// TIA Portal project "ATS Motor Start" (V17)

(* hardware
DEVICE "S7-1200 station_1"  S7-1200 Station
   slot 0: "Rack_0"  S7-1200 Rack  Rack  V1.0
   slot 1: "PLC_2"  CPU 1215C DC/DC/Rly  6ES7 215-1HG40-0XB0  V4.5
*)

// ===== PLC "PLC_2"  CPU 1215C DC/DC/Rly =====

VAR_GLOBAL   // PLC tag table "Default tag table"
   "Clock_Byte" AT %MB0 : Byte;
   "Clock_10Hz" AT %M0.0 : Bool;
   "Clock_5Hz" AT %M0.1 : Bool;
   "Clock_2.5Hz" AT %M0.2 : Bool;
   "Clock_2Hz" AT %M0.3 : Bool;
   "Clock_1.25Hz" AT %M0.4 : Bool;
   "Clock_1Hz" AT %M0.5 : Bool;
   "Clock_0.625Hz" AT %M0.6 : Bool;
   "Clock_0.5Hz" AT %M0.7 : Bool;
   "Tag_1" AT %M2.6 : Bool;
END_VAR

VAR_GLOBAL   // PLC tag table "Tag table_1"
   "emergency_Stop" AT %I0.0 : Bool;
   "Stop" AT %I0.1 : Bool;
   "Start" AT %I0.2 : Bool;
   "PID_Contact" AT %I0.3 : Bool;
   "R1" AT %I0.4 : Bool;
   "R2" AT %I0.5 : Bool;
   "R3" AT %I0.6 : Bool;
   "R4" AT %I0.7 : Bool;
   "R5" AT %I1.0 : Bool;
   "R6" AT %I1.1 : Bool;
   "Thermal_overload" AT %I1.2 : Bool;
   "System_ON" AT %M2.0 : Bool;
   "Backup_supply" AT %Q0.5 : Bool;
   "Main_supply" AT %Q0.6 : Bool;
   "main_k1" AT %Q0.7 : Bool;
   "Star" AT %Q1.0 : Bool;
   "Delta" AT %Q1.1 : Bool;
   "Ats_on" AT %M2.2 : Bool;
   "blue_lamp" AT %Q0.0 : Bool;
   "Green_lamp" AT %Q0.1 : Bool;
   "Red_lamp" AT %Q0.2 : Bool;
   "Yellow_lamp" AT %Q0.3 : Bool;
   "Yellow_lamp_2" AT %Q0.4 : Bool;
   "main_supply_ok" AT %M2.3 : Bool;
   "back_up_ok" AT %M2.4 : Bool;
END_VAR

// folder: System blocks/Program resources

DATA_BLOCK "IEC_Timer_0_DB"   // DB1
{ S7_Optimized_Access := 'TRUE' }
AUTHOR : Simatic
FAMILY : IEC
NAME : IEC_TMR
VERSION : 1.0
// stored: InstanceOfName IEC_TIMER
"IEC_TIMER"
BEGIN
END_DATA_BLOCK

DATA_BLOCK "IEC_Timer_0_DB_2"   // DB3
{ S7_Optimized_Access := 'TRUE' }
AUTHOR : Simatic
FAMILY : IEC
NAME : IEC_TMR
VERSION : 1.0
// stored: InstanceOfName IEC_TIMER
"IEC_TIMER"
BEGIN
END_DATA_BLOCK

DATA_BLOCK "IEC_Timer_0_DB_3"   // DB4
{ S7_Optimized_Access := 'TRUE' }
AUTHOR : Simatic
FAMILY : IEC
NAME : IEC_TMR
VERSION : 1.0
// stored: InstanceOfName IEC_TIMER
"IEC_TIMER"
BEGIN
END_DATA_BLOCK

// folder: (top level)

FUNCTION "Change_over" : Void   // FC1, LAD
{ S7_Optimized_Access := 'TRUE' }
VERSION : 0.1
BEGIN

REGION Network 1: Start system
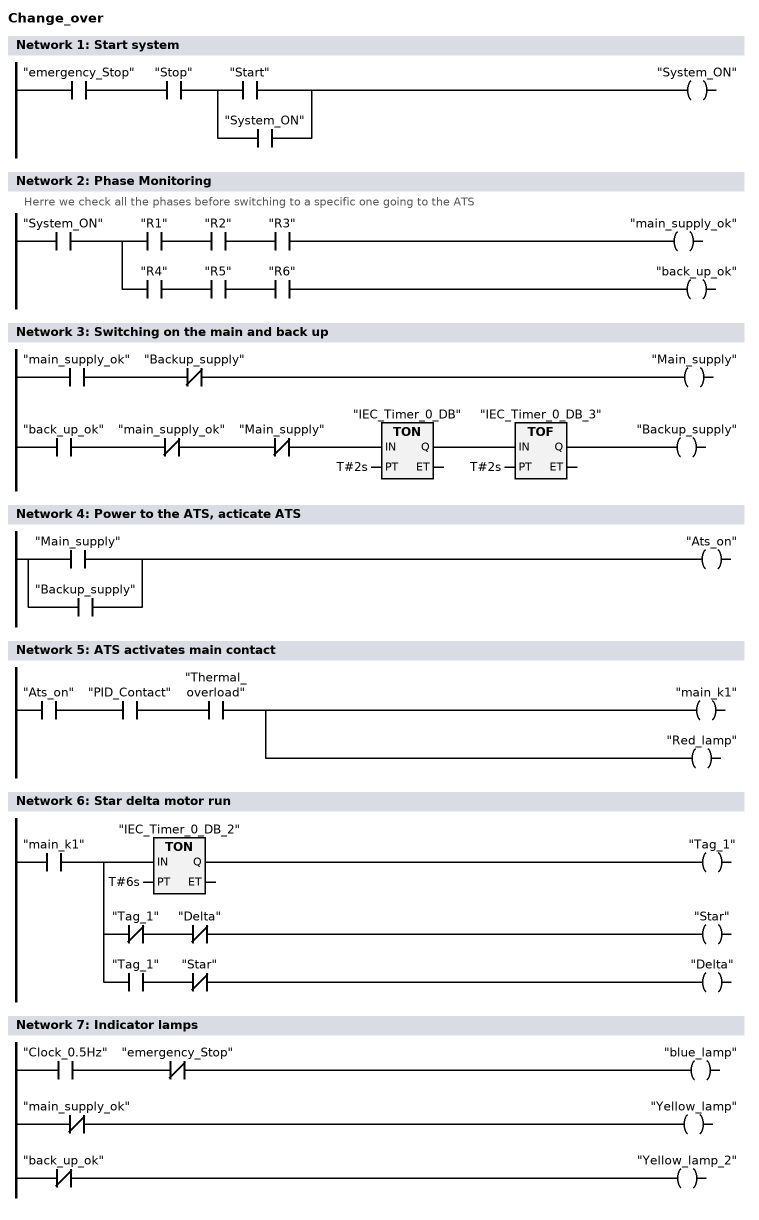
   RUNG wire#powerrail
      Contact( "emergency_Stop" )
      Contact( "Stop" )
      wire#w1
      Contact( "Start" )
      wire#w2
      Coil( "System_ON" )
   END_RUNG
   RUNG wire#w1
      Contact( "System_ON" )
   END_RUNG wire#w2
   // the same network as SCL:
   "System_ON" := "emergency_Stop" AND "Stop" AND ("Start" OR "System_ON");
END_REGION

REGION Network 2: Phase Monitoring
   // Herre we check all the phases before switching to a specific one going to the ATS
   RUNG wire#powerrail
      Contact( "System_ON" )
      wire#w1
      Contact( "R1" )
      Contact( "R2" )
      Contact( "R3" )
      Coil( "main_supply_ok" )
   END_RUNG
   RUNG wire#w1
      Contact( "R4" )
      Contact( "R5" )
      Contact( "R6" )
      Coil( "back_up_ok" )
   END_RUNG
   // the same network as SCL:
   "main_supply_ok" := "System_ON" AND "R1" AND "R2" AND "R3";
   "back_up_ok" := "System_ON" AND "R4" AND "R5" AND "R6";
END_REGION

REGION Network 3: Switching on the main and back up
   "Main_supply" := "main_supply_ok" AND NOT "Backup_supply";
   "IEC_Timer_0_DB".TON(IN := "back_up_ok" AND NOT "main_supply_ok" AND NOT "Main_supply", PT := T#2s);
   "IEC_Timer_0_DB_3".TOF(IN := "IEC_Timer_0_DB".Q, PT := T#2s);
   "Backup_supply" := "IEC_Timer_0_DB_3".Q;
END_REGION

REGION Network 4: Power to the ATS, acticate ATS
   RUNG wire#powerrail
      Contact( "Main_supply" )
      wire#w1
      Coil( "Ats_on" )
   END_RUNG
   RUNG wire#powerrail
      Contact( "Backup_supply" )
   END_RUNG wire#w1
   // the same network as SCL:
   "Ats_on" := "Main_supply" OR "Backup_supply";
END_REGION

REGION Network 5: ATS activates main contact
   RUNG wire#powerrail
      Contact( "Ats_on" )
      Contact( "PID_Contact" )
      Contact( "Thermal_overload" )
      wire#w1
      Coil( "main_k1" )
   END_RUNG
   RUNG wire#w1
      Coil( "Red_lamp" )
   END_RUNG
   // the same network as SCL:
   "main_k1" := "Ats_on" AND "PID_Contact" AND "Thermal_overload";
   "Red_lamp" := "main_k1";
END_REGION

REGION Network 6: Star delta motor run
   "IEC_Timer_0_DB_2".TON(IN := "main_k1", PT := T#6s);
   "Tag_1" := "IEC_Timer_0_DB_2".Q;
   "Star" := "main_k1" AND NOT "Tag_1" AND NOT "Delta";
   "Delta" := "main_k1" AND "Tag_1" AND NOT "Star";
END_REGION

REGION Network 7: Indicator lamps
   RUNG wire#powerrail
      Contact( "Clock_0.5Hz" )
      I_Contact( "emergency_Stop" )
      Coil( "blue_lamp" )
   END_RUNG
   RUNG wire#powerrail
      I_Contact( "main_supply_ok" )
      Coil( "Yellow_lamp" )
   END_RUNG
   RUNG wire#powerrail
      I_Contact( "back_up_ok" )
      Coil( "Yellow_lamp_2" )
   END_RUNG
   // the same network as SCL:
   "blue_lamp" := "Clock_0.5Hz" AND NOT "emergency_Stop";
   "Yellow_lamp" := NOT "main_supply_ok";
   "Yellow_lamp_2" := NOT "back_up_ok";
END_REGION
END_FUNCTION

ORGANIZATION_BLOCK "Main"   // OB1, LAD, ProgramCycle
TITLE = "Main Program Sweep (Cycle)"
{ S7_Optimized_Access := 'TRUE' }
VERSION : 0.1
   VAR_INPUT
      Initial_Call : Bool;   // Initial call of this OB
      Remanence : Bool;   // =True, if remanent data are available
   END_VAR
BEGIN

REGION Network 1
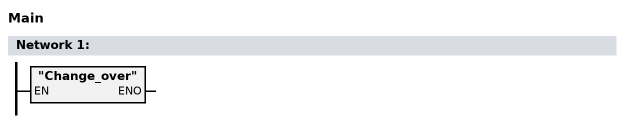
   RUNG wire#powerrail
      "Change_over"()
   END_RUNG
   // the same network as SCL:
   "Change_over"();
END_REGION
END_ORGANIZATION_BLOCK